{attribute 'linkalways'} 
{attribute 'no_explicit_call' := 'This FB is a CLASS and must be accessed using methods or properties'}
{attribute 'enable_dynamic_creation'}
FUNCTION_BLOCK FINAL GT_UDINT EXTENDS Node
VAR
	in1 : _UDINT(0);
	in2 : _UDINT(0);
	out : _BOOL(FALSE);
END_VAR

METHOD PUBLIC Clone : I_Node
VAR
	pNode : POINTER TO GT_UDINT;
END_VAR
pNode := __NEW(GT_UDINT);
Clone := pNode^;
END_METHOD

METHOD FB_init : BOOL
VAR_INPUT
	bInitRetains : BOOL; // if TRUE, the retain variables are initialized (warm start / cold start)
	bInCopyCode : BOOL;  // if TRUE, the instance afterwards gets moved into the copy code (online change)
END_VAR
AddInput('in1',THIS^.in1);
AddInput('in2',THIS^.in2);
AddOutput('out', THIS^.out);
END_METHOD

METHOD PROTECTED OnExecute
VAR
END_VAR
out.Value := in1.Value > in2.Value;
END_METHOD

END_FUNCTION_BLOCK

(* stored: Version 1.1.0.1, ProductVersion 3.1.4024.15
   POU GT_UDINT: Id {b404ed6e-cb7f-426f-96a8-cb9e709380b9}, SpecialFunc None
   Folder Constructor: Id {44999ab8-a23f-45fb-b45d-d8c59336c4c3}
   Method Clone: Id {bcfb8559-b7c6-4eca-a901-a7a874ba79ce}
   Method FB_init: Id {6a08c7b4-815f-40ce-af83-e458978a87a1}
   Method OnExecute: Id {4c0e3307-d5c4-4b1b-92d1-0c59e3bb29db} *)
